INTERFACE ITF_ControlTestWesNiek

PROPERTY HMIDepalletizerCurrentState : E_PackMLStates
GET
END_GET
SET
END_SET
END_PROPERTY

PROPERTY HMIKlaarVoorInvoer : BOOL
GET
END_GET
SET
END_SET
END_PROPERTY

PROPERTY HMIKlaarVoorUitvoer : BOOL
GET
END_GET
SET
END_SET
END_PROPERTY

PROPERTY HMILiftAanUit : BOOL
GET
END_GET
SET
END_SET
END_PROPERTY

PROPERTY HMIMotorSchuifStatus : E_MotorZuigSchuifStatus
GET
END_GET
SET
END_SET
END_PROPERTY

PROPERTY HMIMotorZuigStatus : E_MotorZuigSchuifStatus
GET
END_GET
SET
END_SET
END_PROPERTY

PROPERTY HMIPinnenUitYesNo : BOOL
GET
END_GET
SET
END_SET
END_PROPERTY

PROPERTY HMIRolbandAanUit : BOOL
GET
END_GET
SET
END_SET
END_PROPERTY

END_INTERFACE

(* stored: Version 1.1.0.1
   Itf ITF_ControlTestWesNiek: Id {649c8754-d58c-4c47-a718-f4ea8576dd07}
   Folder HMIDepalletizer: Id {997b8582-d383-4605-97f3-6c83282cb7ee}
   Property HMIDepalletizerCurrentState: Id {0ef3e29f-48aa-47b7-a5ce-7e52534533a3}
   Get Get: Id {44c9355d-12cd-4dd0-a2c3-140a0ca4ecb0}
   Set Set: Id {f8588cc0-52a7-415a-ae9d-883a7735beff}
   Property HMIKlaarVoorInvoer: Id {4be0e5f1-2cf7-4ae8-8288-a8d84ce840ab}
   Get Get: Id {bc735157-6c15-468c-881e-fb3321376b62}
   Set Set: Id {ef98c771-acb1-4cbd-bb77-26f31ee886d9}
   Property HMIKlaarVoorUitvoer: Id {b821f182-8226-4bc9-bab9-24dc0e3f4a57}
   Get Get: Id {c7404342-cb2e-4b30-8c13-d982bf95b7fd}
   Set Set: Id {e485a1d8-b46d-4e09-8aeb-645deae30f1f}
   Property HMILiftAanUit: Id {ffba2307-5455-4f89-b95c-731ed3633573}
   Get Get: Id {5c99a85a-dca1-4fd5-825d-8d702237016d}
   Set Set: Id {96917651-9a2e-4dfe-ba9c-fe25e61d34f9}
   Property HMIMotorSchuifStatus: Id {93b4d50d-0133-4eb2-b5dd-e3afa33e9b41}
   Get Get: Id {31f888ff-2d92-4273-9c85-a0798e5c8d3f}
   Set Set: Id {b8765be3-2151-4250-90e1-b3f0da3472c2}
   Property HMIMotorZuigStatus: Id {4fd9bfa6-0362-4998-b829-87154b6bb0a3}
   Get Get: Id {78720a31-3c24-4304-a680-698b968b8f25}
   Set Set: Id {9e2faccf-cab5-4b81-be1b-a857cffe1038}
   Property HMIPinnenUitYesNo: Id {2a3cff79-4fc7-4cf9-8754-a72f5540bb84}
   Get Get: Id {d4bac406-4082-424b-8a18-ba7b83fae055}
   Set Set: Id {17aceb82-828d-4ca8-b05d-18ee02f03a8b}
   Property HMIRolbandAanUit: Id {9090e5b2-e364-4d06-80c5-f357c562fdea}
   Get Get: Id {07cc6c29-0b75-449e-a463-5d7e94f44c31}
   Set Set: Id {2181057f-2073-4afa-892d-8591fed4b9c2} *)
